// TIA Portal V19 export
VAR_GLOBAL   // PLC tag table "STEP7 classic symbols"
   "hf LyeOnly" AT %I600.1 : Bool;   // info for CIP process (Not used)
   hfOperationsMode AT %IW622 : Int;   // IMA Hassia - operations mode,0=shutdown,1=CIP, 2=SIP,4=Production,8=Adjustments
   prProductAvailableF1 AT %Q608.0 : Bool;   // product for filler 1 is ready
   "A02-ACID CONTAINER EMPTY" AT %M70.1 : Bool;   // ALARM 2
   "A19-TT 01.63 TOO LOW" AT %M72.2 : Bool;   // ALARM 19
   "A36-FB FAULT VALVE 01.15" AT %M74.3 : Bool;   // ALARM 36
   "A55-CIP UNIT OCCUIPED" AT %M76.6 : Bool;   // ALARM 55
   "AutoTT0172/IP0157" AT %M91.0 : Bool;   // REGULATOR TT01.72/IP01.57 IN AUTO MODE
   CIP_Hamba_bit_06 AT %M150.6 : Bool;
   CT_ACID_OK AT %M32.4 : Bool;   // ACID CONCENTRATION WITHIN LIMITS
   "DUMMY TEST AIR" AT %M98.5 : Bool;   // DUMMY TEST AIR SUPPLY
   HSL0165_Proxy AT %M50.1 : Bool;
   P_IP0157 AT %QW274 : Word;   // Steam regulating valve
   "Last Scan Time" AT %MW40 : Int;   // Previous Scan Time
   "M21.1" AT %M21.1 : Bool;
   MY0108 AT %M247.3 : Bool;   // Q 9.3; Output modul 1 Channel 11
   MY0147 AT %M248.7 : Bool;   // Q 20.7; Output modul 2 Channel 7
   MY0911 AT %M253.2 : Bool;
   M_LP_Steam_ON AT %M254.6 : Bool;
   One_shut_on AT %M152.3 : Bool;
   P_PT0167 AT %IW266 : Word;   // Filling pressure
   Product_Route AT %Q41.6 : Bool;   // Hamba
   "R.NOT USED 9" AT %M245.0 : Bool;   // RECIEVE FROM UHT MPI NET, NOT USED
   "S.T.02.TANK PRESELE." AT %M243.5 : Bool;   // TANK 2 PRESELECTED SEND TO UHT FROM TANK 02.00 MPI NET
   "S1 STOP PRODUCTION TANK" AT %M113.1 : Bool;   // STEP 1 STOP PRODUCTION TANK
   "S17 FILLER" AT %M126.1 : Bool;   // STEP 17 FILLER
   "S23 FILLER" AT %M126.7 : Bool;   // STEP 23 FILLER
   "S34 FILLER" AT %M128.2 : Bool;   // STEP 34 FILLER
   "S46 FILLER" AT %M129.6 : Bool;   // STEP 46 FILLER
   "S9 CIP TANK" AT %M119.1 : Bool;   // STEP 9 CIP
   SIP_Hamba_bit_05 AT %M151.5 : Bool;
   ST_CIP_M0139 AT %M138.0 : Bool;   // START CIP PUMP
   Sterilisation_Steam AT %Q41.3 : Bool;   // Hamba
   "T 37 DELAY TT 01.78" AT %T37 : Timer;   // DELAY ALARM TT 01.78 AS BARRIER
   "T53 DETERGENT CONC OK" AT %T53 : Timer;   // DETERGENT CONCENTRATION OK IN X SECONDS
   "TEST BARRIERS" AT %M94.3 : Bool;   // TEST TEMPERATURES AS BARRIERES
   TIM20 AT %M61.2 : Bool;   // START TIMER 20
   TIM37 AT %M63.3 : Bool;   // START TIMER 37
   TIM54 AT %M65.4 : Bool;   // START TIMER 54
   "UHT_STERILE?" AT %I25.5 : Bool;   // UHT STERILE
   Y0104S AT %I12.2 : Bool;   // FEEDBACK SET VALVE 01.04
   Y0114R AT %I16.7 : Bool;   // FEEDBACK RESET VALVE 01.14
   Y0137 AT %Q20.4 : Bool;   // WATER TO CONDENSATER VALVE
   Y0905R AT %I45.1 : Bool;   // On off valve
   Y0910 AT %Q40.6 : Bool;   // Routing valve
   "0.5Hz" AT %M10.7 : Bool;   // CYCLIC CLOCK
   "A04-TANK NOT CLEAN" AT %M70.3 : Bool;   // ALARM 4
   "A21-TT 01.76 LOW" AT %M72.4 : Bool;   // ALARM 21
   "A38-FB FAULT MOTOR 01.30" AT %M74.5 : Bool;   // ALARM 38
   ACID_READY AT %Q29.0 : Bool;   // ACID READY
   ATI AT %M11.2 : Bool;   // Always true input
   "B01.41" AT %I17.4 : Bool;   // HIGH LEVEL ELECTRODE CIP TANK
   CAUSTIC_REQ AT %I33.2 : Bool;   // CAUSTIC REQUIRED
   "CIP_OCCUIPED?" AT %I25.7 : Bool;   // CIP OCCUPIED
   "DUMMY TEST STEAM" AT %M98.4 : Bool;   // DUMMY TEST STEAM SUPPLY
   "I33.7SPARE" AT %I33.7 : Bool;   // SPARE
   M0139 AT %Q9.1 : Bool;   // CIP PUMP
   "M21.3" AT %M21.3 : Bool;   // fp bit for depressurise pg line if not sterile
   MY0111 AT %M246.4 : Bool;   // Q 8.4; Output modul 1 Channel 4
   MY0158 AT %M249.1 : Bool;   // Q 21.1; Output modul 2 Channel 9
   "M_251.3SpareOutput" AT %M251.3 : Bool;   // Q 29.3; Output modul 3 Channel 11
   M_PACK2 AT %M249.4 : Bool;   // Q 21.4; Output modul 2 Channel 12
   Min_F2 AT %IW618 : Word;
   "PULSE 01.13 CIP" AT %M94.6 : Bool;   // PULSE VALVE 01.13 IN CIP
   Prod_Hamba_bit_00 AT %M153.0 : Bool;
   "Q537.0" AT %Q537.0 : Bool;   // Polygon Filler 2 EOL in Use Becon
   "R.UHT STERIL/PRESTE" AT %M244.0 : Bool;   // UHT STERIL/PRESTERIL. RECIEVE FROM UHT MPI NET
   RTE_404_TestBit AT %M19.0 : Bool;   // for testing RTE 404
   "S0 CHAIN WASH" AT %M137.0 : Bool;   // STEP 0 CHAIN WASH
   "S10 CIP TANK" AT %M119.2 : Bool;   // STEP 10 CIP
   "S18 FILLER" AT %M126.2 : Bool;   // STEP 18 FILLER
   "S25 FILLER" AT %M127.1 : Bool;   // STEP 25 FILLER
   "S36 FILLER" AT %M128.4 : Bool;   // STEP 36 FILLER
   "S48 FILLER" AT %M130.0 : Bool;   // STEP 48 FILLER
   SCADA_WD AT %MW200 : Int;   // SCADA Watch Dog
   SIP_Hamba_bit_07 AT %M151.7 : Bool;
   "T 14 STERILE TIME" AT %T14 : Timer;   // STERILIZING TIME ASEPTIC TANK
   "T 39 RUN 01.30" AT %T39 : Timer;   // RUN TIME AGITATOR 01.30
   "T55 ACID DOSING TOO LONG" AT %T55 : Timer;   // ACID DOSING TIME TOO LONG, SEARCH FOR FAILURE
   "TEST FILLING PRESSURE" AT %M94.4 : Bool;   // TEST FILLING PRESSURE
   TIM22 AT %M61.4 : Bool;   // START TIMER 22
   TIM39 AT %M63.5 : Bool;   // START TIMER 39
   TIM56 AT %M65.6 : Bool;   // START TIMER 56
   "UPD.TIMER 14" AT %M84.0 : Bool;   // UPDATE STERILE TIMER
   "V0945-SV2 DelayOff" AT %T77 : Timer;   // V0945-SV2 DelayOff (Production Only)
   WATER_SUPPLY_PUMP AT %Q29.2 : Bool;   // WATER PUMP
   Y0108R AT %I17.3 : Bool;   // FEEDBACK RESET VALVEL 01.08
   Y0115 AT %Q9.0 : Bool;   // WATER TO BALANCE TANK VALVE
   Y0144 AT %Q20.6 : Bool;   // DRAIN VALVE CIP 01.01
   Y0906 AT %Q40.2 : Bool;   // Routing valve
   Y0910S AT %I44.6 : Bool;   // Routing valve
   "hf PreRinse1" AT %I601.0 : Bool;   // prerinse 1
   mw212_DW AT %MW212 : Word;   // Dummy word for fc3
   "hf HoperLevelF1" AT %IW610 : Int;   // Hassia Filler 1 Hopper Level (1000 x 0.1 = 100.0%)
   "hf SIPrequest" AT %I604.0 : Bool;   // request sterilization
   prF2_AhvLevel AT %QW610 : Int;   // Supplying AHV Level for IMA Hassia- Filler2
   "2Hz" AT %M10.3 : Bool;   // CYCLIC CLOCK
   "A14-WAITING FOR CIPUNIT" AT %M71.5 : Bool;   // ALARM 14
   "A31-FB FAULT VALVE 01.09" AT %M73.6 : Bool;   // ALARM 31
   "A48-FB FAULT VALVE 01.19" AT %M75.7 : Bool;   // ALARM 48
   AHV_SHUT_DOWN AT %Q28.3 : Bool;   // AHV SHUT DOWN
   CIP_Hamba_bit_01 AT %M150.1 : Bool;
   "DUMMY 2 FILLING" AT %M100.1 : Bool;   // DUMMY USED IN FILLING
   DisableMonitoringTT0951 AT %M152.2 : Bool;
   "FILLING PIPE DRAINED" AT %M95.2 : Bool;   // FILLING PIPE DRAINED INITIAL START
   GS22_62 AT %I46.1 : Bool;
   "I      47.3" AT %I47.3 : Bool;
   "M20.2" AT %M20.2 : Bool;   // acDataPointer_FIFO #busy in/out
   MW_202 AT %MW202 : Word;
   MY0135 AT %M248.2 : Bool;   // Q 20.2; Output modul 2 Channel 2
   "MY0906 Cycle On" AT %M253.6 : Bool;
   M_Barrier_Sterlising AT %M254.5 : Bool;
   M_WATER_SUPPLY_PUMP AT %M251.2 : Bool;   // Q 29.2; Output modul 3 Channel 10
   PROG_2_SELECTED AT %I32.7 : Bool;   // PROGRAM 2 SELECTED
   Prod_Hamba_bit_10 AT %M154.2 : Bool;
   "R.NOT USED 15" AT %M245.6 : Bool;   // RECIEVE FROM UHT MPI NET, NOT USED
   RINSE_REQ AT %I33.1 : Bool;   // RINSE REQUIRED
   "S.T.02.NOT USED 7" AT %M243.6 : Bool;   // SEND TO UHT FROM TANK 02.00 MPI NET, NOT USED
   "S1 CIP TANK" AT %M118.1 : Bool;   // STEP 1 CIP
   "S15 CIP TANK" AT %M119.7 : Bool;   // STEP 15 CIP
   "S2 TOTAL STOP TANK" AT %M114.2 : Bool;   // STEP 2 TOTAL STOP TANK
   "S3 STOP PRESTE. TANK" AT %M109.3 : Bool;   // STEP 3 STOP PRESTERILIZING TANK
   "S41 FILLER" AT %M129.1 : Bool;   // STEP 41 FILLER
   "S7 CIP TANK" AT %M118.7 : Bool;   // STEP 7 CIP
   SIP_Hamba_bit_00 AT %M151.0 : Bool;
   "Spare m254.7" AT %M254.7 : Bool;
   "T 32 ACID CIRCULATION" AT %T32 : Timer;   // CIRCULATING ACID ASEPTIC TANK
   "T 49 OPEN 01.08 CIP" AT %T49 : Timer;   // OPEN VALVE 01.08 CIP
   "TANK STERILE" AT %M90.2 : Bool;   // TANK IS STERILE
   TIM15 AT %M60.5 : Bool;   // START TIMER 15
   TIM32 AT %M62.6 : Bool;   // START TIMER 32
   TIM49 AT %M64.7 : Bool;   // START TIMER 49
   P_TT0178 AT %IW258 : Word;   // Steam barrier filling valve
   "Trigger bit 4" AT %M14.3 : Bool;   // Trigger bit for calls in item control
   "UPD.TIMER 33" AT %M85.2 : Bool;   // UPDATE WATER 3 TIMER
   ValveHandling3 AT %M3.7 : Bool;   // VALVE HANDLING
   Y0103 AT %Q8.1 : Bool;   // CIP / STEAM INLET VALVE
   Y0112S AT %I12.5 : Bool;   // FEEDBACK SET VALVE 01.12
   Y0119 AT %Q20.0 : Bool;   // FLUSH CHAIN WASH
   Y0904 AT %Q40.0 : Bool;   // On off valve
   "A12-DRAIN TANK NOT ALLOW" AT %M71.3 : Bool;   // ALARM 12
   "A29-FB FAULT VALVE 01.03" AT %M73.4 : Bool;   // ALARM 29
   "A46-FB FAULT VALVE 01.17" AT %M75.5 : Bool;   // ALARM 46
   Barrier_Sterile AT %Q41.5 : Bool;   // Hamba
   DUMMY_ALARM AT %M11.4 : Bool;   // Dummy USED FOR ALARMS ETC
   FILLER_ON_PROD AT %I32.4 : Bool;   // FILLER ON PRODUCT
   "I      47.1" AT %I47.1 : Bool;
   MY0119 AT %M248.0 : Bool;   // Q 20.0; Output modul 2 Channel 0
   MY0905 AT %M252.4 : Bool;
   M_AHV_STERILE AT %M250.4 : Bool;   // Q 28.4; Output modul 3 Channel 4
   M_TANK_READY AT %M251.6 : Bool;   // Q 29.6; Output modul 3 Channel 14
   PROD_AVAILABLE AT %Q28.5 : Bool;   // PRODUCT AVAILABLE
   Prod_Hamba_bit_08 AT %M154.0 : Bool;
   "R.NOT USED 13" AT %M245.4 : Bool;   // RECIEVE FROM UHT MPI NET, NOT USED
   "Request CIP Pump ON" AT %I33.6 : Bool;   // SPARE
   "S.T.01.TANK READY" AT %M242.4 : Bool;   // TANK 1 READY SEND TO UHT FROM TANK 01.00 MPI NET
   "S0 TOTAL STOP TANK" AT %M114.0 : Bool;   // MAIN FLAG TOTAL STOP TANK
   "S14 CIP TANK" AT %M119.6 : Bool;   // STEP 14 CIP
   "S2 STOP PRESTE. TANK" AT %M109.2 : Bool;   // STEP 2 STOP PRESTERILIZING TANK
   "S3 PRESTERILIZING" AT %M110.3 : Bool;   // STEP 3 PRESTERILIZING TANK
   "S4 STOP CIP TANK" AT %M122.4 : Bool;   // STEP 4 STOP CIP
   "S6 FILLER" AT %M124.6 : Bool;   // STEP 06 FILLER
   SIP_Hamba_High_SteamPres AT %M152.0 : Bool;
   "T 30 WATER 2" AT %T30 : Timer;   // INTERMEDIATE RINSE ASEPTIC TANK
   "T 47 OPEN 01.13 PRES" AT %T47 : Timer;   // OPEN TIME VALVE 01.13 IN PRESTERILIZING
   "TANK CLEAN" AT %M0.1 : Bool;   // TANK IS CLEAN
   TIM13 AT %M60.3 : Bool;   // START TIMER 13
   TIM30 AT %M62.4 : Bool;   // START TIMER 30
   TIM47 AT %M64.5 : Bool;   // START TIMER 47
   TIM64 AT %M66.6 : Bool;   // START TIMER 64
   P_TT0172 AT %IW262 : Word;   // CIP temperature
   "Trigger bit 2" AT %M14.1 : Bool;   // Trigger bit for calls in item control
   "UPD.TIMER 31" AT %M85.0 : Bool;   // UPDATE DOSING ACID TIMER
   ValveHandling1 AT %M2.4 : Bool;   // VALVE HANDLING
   Y0101R AT %I16.0 : Bool;   // FEEDBACK RESET VALVE 01.01
   Y0112 AT %Q8.5 : Bool;   // FILLING LINE STOP VALVE
   Y0117S AT %I24.1 : Bool;   // FEEDBACK SET VALVE 01.17
   Y0902 AT %Q29.4 : Bool;   // Low steam pressure
   Y0907S AT %I44.3 : Bool;   // On off valve
   "hf HoperLevelF2" AT %IW612 : Int;   // Hassia Filler 2 Hopper Level (1000 x 0.1 = 100.0%)
   "hf SIPrunning" AT %I604.1 : Bool;   // sterilization is running
   "prLife bit" AT %Q600.0 : Bool;   // check communication (clocked signal 0,5 Hz)
   prEnableCIPValveFlipsF1 AT %Q601.1 : Bool;
   "1HZ_ONESHOT" AT %M11.0 : Bool;
   "A10-TANK IS BEEING FILL." AT %M71.1 : Bool;   // ALARM 10
   "A27-SIEMENS BATTERY LOW" AT %M73.2 : Bool;   // ALARM 27
   "A44-FB FAULT VALVE 02.38" AT %M75.3 : Bool;   // ALARM 44
   AHV_CLOSED AT %Q28.0 : Bool;   // AHV BARRIER CLOSED
   CIP_Running AT %I24.6 : Bool;   // Hamba
   "DUMMY1 DRAIN" AT %M98.7 : Bool;   // DUMMY DRAIN FILLING PIPE
   FILLER_2_OK AT %I32.5 : Bool;   // FILLER 2 BARRIER TEMP. OK
   ForceValves AT %M12.0 : Bool;   // FORCE VALVES TO AUTO
   "I      46.7" AT %I46.7 : Bool;
   MANUAL AT %M3.3 : Bool;   // VALVE HANDLING
   MY0117 AT %M247.4 : Bool;   // Q 9.4; Output modul 1 Channel 12
   MY0903 AT %M252.2 : Bool;
   M_AHV_READY AT %M250.2 : Bool;   // Q 28.2; Output modul 3 Channel 2
   M_Sip_Steam AT %M254.1 : Bool;
   PACK2 AT %Q21.4 : Bool;   // RELAY SIGNAL TO PACKING PRODUCT AVAILA.
   Prod_Hamba_bit_06 AT %M153.6 : Bool;
   "R.NOT USED 11" AT %M245.2 : Bool;   // RECIEVE FROM UHT MPI NET, NOT USED
   "S.T.01.TANK OPEN" AT %M242.3 : Bool;   // TANK 1 OPEN SEND TO UHT FROM TANK 01.00 MPI NET
   "S0 STOP PRESTE. TANK" AT %M109.0 : Bool;   // MAIN FLAG STOP PRESTERILIZING TANK
   "S13 CIP TANK" AT %M119.5 : Bool;   // STEP 13 CIP
   "S2 PRESTERILIZING" AT %M110.2 : Bool;   // STEP 2 PRESTERILIZING TANK
   "S3 CIP TANK" AT %M118.3 : Bool;   // STEP 3 CIP
   "S4 FILLER" AT %M124.4 : Bool;   // STEP 04 FILLER
   "S6 CHAIN WASH" AT %M137.6 : Bool;   // STEP 6 CHAIN WASH
   "T 28 DOSING LYE" AT %T28 : Timer;   // DOSING LYE ASEPTIC TANK
   "T 45 PURGE" AT %T45 : Timer;   // PURGING FILLING PIPE
   T83 AT %T83 : Timer;   // delay close V0945 after flips
   TIM11 AT %M60.1 : Bool;   // START TIMER 11
   TIM28 AT %M62.2 : Bool;   // START TIMER 28
   TIM45 AT %M64.3 : Bool;   // START TIMER 45
   TIM62 AT %M66.4 : Bool;   // START TIMER 62
   TRIGGERBYTE AT %MB14 : Byte;   // USED FOR OUTPUT HANDLER
   "UPD.TIMER 29" AT %M84.6 : Bool;   // UPDATE LYE CIRCULATION TIMER
   X0913 AT %Q41.7 : Bool;   // Cip lamp
   Y0111R AT %I16.4 : Bool;   // FEEDBACK RESET VALVE 01.11
   Y0117 AT %Q9.4 : Bool;   // CIP
   Y0545 AT %Q21.2 : Bool;   // STEAM BY-PASS VALVE REDUCED
   Y0907 AT %Q40.3 : Bool;   // On off valve
   Y0912S AT %I25.3 : Bool;   // SPARE
   "hf DrainMachine" AT %I601.1 : Bool;   // drain machine
   Y0910R AT %I45.6 : Bool;   // Routing valve
   "hf NoTimeStop" AT %I600.4 : Bool;   // no fault and no stop during CIP at Hassia Machine
   mw210_DW AT %MW210 : Word;   // Dummy word for fc3
   prSIPRunningF2 AT %Q604.2 : Bool;   // information product line filler 2 SIP is running
   "A06-NO STEAM" AT %M70.5 : Bool;   // ALARM 6
   "A23-NO WATER" AT %M72.6 : Bool;   // ALARM 23
   "A40-LYE DOSING TOO LONG" AT %M74.7 : Bool;   // ALARM 40
   ACTIVATE AT %M3.4 : Bool;   // VALVE HANDLING
   "B01.65" AT %I17.6 : Bool;   // HIGH LEVEL ELECTRODE STERILE TANK
   CHANGING AT %M2.3 : Bool;   // VALVE HANDLING
   CIP_PROG_2 AT %M135.2 : Bool;   // PROGRAM SELECT 2 CIP FILLER
   "DUMMY TEST TT 01.78" AT %M98.3 : Bool;   // DUMMY TEST TT 01.78 AS BARRIER
   "M21.5" AT %M21.5 : Bool;   // PG line Sterile memory
   MY0113 AT %M246.6 : Bool;   // Q 8.6; Output modul 1 Channel 6
   MY0238 AT %M247.7 : Bool;   // Q 9.7; Output modul 1 Channel 15
   "M_251.5SpareOutput" AT %M251.5 : Bool;   // Q 29.5; Output modul 3 Channel 13
   M_ProdLineBeingCleaned AT %M249.5 : Bool;   // Q 21.5; Output modul 2 Channel 13 was M_PACK3
   Prod_Hamba_bit_02 AT %M153.2 : Bool;
   "R.Acid Level Ok" AT %M244.7 : Bool;   // RECIEVE FROM UHT MPI NET, NOT USED
   RTE_405_TestBit AT %M19.1 : Bool;
   "S.T.01.NOT USED 7" AT %M242.6 : Bool;   // SEND TO UHT FROM TANK 01.00 MPI NET, NOT USED
   "S0 FILLER" AT %M124.0 : Bool;   // STEP 00 MAIN FILLER
   "S11 CIP TANK" AT %M119.3 : Bool;   // STEP 11 CIP
   "S19 FILLER" AT %M126.3 : Bool;   // STEP 19 FILLER
   "S27 FILLER" AT %M127.3 : Bool;   // STEP 27 FILLER
   "S38 FILLER" AT %M128.6 : Bool;   // STEP 38 FILLER
   "S5 CHAIN WASH" AT %M137.5 : Bool;   // STEP 5 CHAIN WASH
   "SPIN 01.30 CIP" AT %M94.5 : Bool;   // SPIN AGITATOR IN CIP
   "T 16 BLOW OUT COND" AT %T16 : Timer;   // BLOW OUT CONDENSATE
   "T 41 DELAY STEAM" AT %T41 : Timer;   // DELAY ALARM STEAM
   "T61 CLOSE Y0101" AT %T61 : Timer;   // DELAY BETWEEN Y0101 AND Y0124 (CLOSE)
   TIM24 AT %M61.6 : Bool;   // START TIMER 24
   TIM41 AT %M63.7 : Bool;   // START TIMER 41
   TIM58 AT %M66.0 : Bool;   // START TIMER 58
   "UPD.TIMER 16" AT %M84.2 : Bool;   // UPDATE BLOW OUT CONDENSATE TIMER
   Y0109 AT %Q8.3 : Bool;   // COOLING WATER TO JACKET VALVE
   Y0115S AT %I13.0 : Bool;   // FEEDBACK SET VALVE 01.15
   Y0148 AT %Q21.0 : Bool;   // STEAM VALVE TO STERILZING
   "hf MachineSterile" AT %I604.2 : Bool;   // machine sterile
   "m20.0" AT %M20.0 : Bool;   // FP
   prSIPRunningF1 AT %Q604.1 : Bool;   // information product line filler 1 SIP is running
   "0.625Hz" AT %M10.6 : Bool;   // CYCLIC CLOCK
   "A05-NO INSTRUMENT AIR" AT %M70.4 : Bool;   // ALARM 5
   "A22-TT 01-78 LOW" AT %M72.5 : Bool;   // ALARM 22
   "A39-TANK READY FOR PROD" AT %M74.6 : Bool;   // ALARM 39
   ACID_REQ AT %I33.3 : Bool;   // ACID REQUIRED
   AcidCipPressure AT %M96.3 : Bool;
   "B01.42" AT %I17.5 : Bool;   // LOW LEVEL ELECTRODE CIP TANK
   CHAIN_WASH AT %I33.4 : Bool;   // CHAIN WASH
   CIP_PROG_1 AT %M135.1 : Bool;   // PROGRAM SELECT 1 CIP FILLER
   "DUMMY TEST TT 01.76" AT %M98.2 : Bool;   // DUMMY TEST TT 01.76 AS BARRIER
   "Hamba FP1 Route OK" AT %M104.1 : Bool;
   "I553.0" AT %I533.0 : Bool;   // M0941 - Running (M0940 Cooling Fan)
   Init_Scan AT %M0.0 : Bool;   // First Scan
   M0139S AT %I13.1 : Bool;   // FEEDBACK MOTOR 01.39 RUNNING
   "M21.4" AT %M21.4 : Bool;   // depressurise pg line if clean not sterile
   MY0112 AT %M246.5 : Bool;   // Q 8.5; Output modul 1 Channel 5
   MY0237 AT %M247.6 : Bool;   // Q 9.6; Output modul 1 Channel 14
   "M_251.4SpareOutput" AT %M251.4 : Bool;   // Q 29.4; Output modul 3 Channel 12
   M_PROD_AVAILABLE AT %M250.5 : Bool;   // Q 28.5; Output modul 3 Channel 5
   "PULSE 01.18 PRESTERILI" AT %M94.0 : Bool;   // PULSING VALVE 01.13 IN PRESTERILIZING
   Prod_Hamba_bit_01 AT %M153.1 : Bool;
   "Q537.1" AT %Q537.1 : Bool;   // Polygon F2 Product at Filler
   "S.T.01.ALARM PULS" AT %M242.2 : Bool;   // ALARM PULS SEND TO UHT FROM TANK 01.00 MPI NET
   "S0 CIP TANK" AT %M118.0 : Bool;   // MAIN FLAG CIP
   "S10 FILLER" AT %M125.2 : Bool;   // STEP 10 FILLER
   "S19 CIP TANK" AT %M120.3 : Bool;   // STEP 19 CIP
   "S26 FILLER" AT %M127.2 : Bool;   // STEP 26 FILLER
   "S37 FILLER" AT %M128.5 : Bool;   // STEP 37 FILLER
   "S49 FILLER" AT %M130.1 : Bool;   // STEP 49 FILLER
   "SOFTKEY 5 DRAIN TANK" AT %M99.6 : Bool;   // SOFTKEY START DRAIN TANK
   "T 15 COOLING TIME" AT %T15 : Timer;   // COOLING TIME ASEPTIC TANK
   "T 40 RESET STOP LIGHT" AT %T40 : Timer;   // DELAY RESET STOP LIGHT AFTER 3 SEC
   "T60 OPEN Y0101" AT %T60 : Timer;   // DELAY BETWEEN Y0124 AND Y0101 (OPEN)
   TIM23 AT %M61.5 : Bool;   // START TIMER 23
   TIM40 AT %M63.6 : Bool;   // START TIMER 40
   TIM57 AT %M65.7 : Bool;   // START TIMER 57
   "UPD.TIMER 15" AT %M84.1 : Bool;   // UPDATE COOLING TIMER
   Y0108S AT %I13.3 : Bool;   // FEEDBACK SET VALVEL 01.18
   Y0115R AT %I17.0 : Bool;   // FEEDBACK RESET VALVE 01.15
   Y0147 AT %Q20.7 : Bool;   // STEAM VALVE TO 01.13
   "Y0906 Cycle Off" AT %M253.7 : Bool;
   Y0911 AT %Q40.7 : Bool;   // On off valve
   "A01-LYE CONTAINER EMPTY" AT %M70.0 : Bool;   // ALARM 1
   "A18-TT 01.60 TOO LOW" AT %M72.1 : Bool;   // ALARM 18
   "A35-FB FAULT VALVE 01.14" AT %M74.2 : Bool;   // ALARM 35
   "A54-NO CIP PROG SEL" AT %M76.5 : Bool;   // ALARM 54
   "AutoPT0167/IP0149" AT %M91.2 : Bool;   // REGULATOR PT01.67/IP01.49 IN AUTO MODE
   CIP_Hamba_bit_05 AT %M150.5 : Bool;
   P_CT0182 AT %IW270 : Word;   // CIP Contration return
   "DUMMY START AGITATOR" AT %M99.3 : Bool;   // DUMMY START AGITATOR
   "FS01.81" AT %I13.2 : Bool;   // FLOW SWITCH CIP RETURN
   "I      47.7" AT %I47.7 : Bool;
   P_IP014950 AT %QW272 : Word;   // Sterile air control valves
   "M21.0" AT %M21.0 : Bool;
   MY0104 AT %M246.2 : Bool;   // Q 8.2; Output modul 1 Channel 2
   MY0144 AT %M248.6 : Bool;   // Q 20.6; Output modul 2 Channel 6
   MY0910 AT %M253.1 : Bool;
   M_Cip_Route AT %M254.0 : Bool;
   Max_F2 AT %IW620 : Word;
   One_shut_off AT %M152.4 : Bool;
   Product_Request AT %I24.5 : Bool;   // Hamba
   "R.NOT USED 6" AT %M244.5 : Bool;   // RECIEVE FROM UHT MPI NET, NOT USED
   RTE_404_Cip_Route_Open AT %M255.0 : Bool;   // Allow Gemini Route 411 and Tankroom Route 404_405 to Run
   "S.T.02.TANK OPEN" AT %M243.3 : Bool;   // TANK 2 OPEN SEND TO UHT FROM TANK 02.00 MPI NET
   "S1 STOP PRESTE. TANK" AT %M109.1 : Bool;   // STEP 1 STOP PRESTERILIZING TANK
   "S17 CIP TANK" AT %M120.1 : Bool;   // STEP 17 CIP
   "S22 FILLER" AT %M126.6 : Bool;   // STEP 22 FILLER
   "S33 FILLER" AT %M128.1 : Bool;   // STEP 33 FILLER
   "S45 FILLER" AT %M129.5 : Bool;   // STEP 45 FILLER
   "S8 FILLER" AT %M125.0 : Bool;   // STEP 08 FILLER
   SIP_Hamba_bit_04 AT %M151.4 : Bool;
   StepOldStatus AT %MW208 : Word;   // Dummy word for fc3
   "T 36 DELAY TT 01.76" AT %T36 : Timer;   // DELAY ALARM TT 01.76 AS BARRIER
   T20_Trigger_bit AT %T20 : Timer;
   "TBM DUMMY MOTOR 01.39" AT %M79.0 : Bool;   // DUMMY FEED-BACK FOR RESET
   TIM19 AT %M61.1 : Bool;   // START TIMER 19
   TIM36 AT %M63.2 : Bool;   // START TIMER 36
   TIM53 AT %M65.3 : Bool;   // START TIMER 53
   "Trigger bit 8" AT %M14.7 : Bool;   // Trigger bit for calls in item control
   UnforceValves AT %M12.1 : Bool;   // UNFORCE VALVES FROM AUTO
   Y0104R AT %I16.2 : Bool;   // FEEDBACK RESET VALVE 01.04
   Y0114 AT %Q8.7 : Bool;   // CIP RETURN / DRAIN VALVE
   Y0136 AT %Q20.3 : Bool;   // STEAM TO CONDENSTATE VALVE
   Y0905 AT %Q40.1 : Bool;   // On off valve
   Y0909S AT %I44.5 : Bool;   // On off valve
   "hf MachineIsClean" AT %I601.7 : Bool;   // machine is clean
   "m19.3" AT %M19.3 : Bool;   // Tank Sterile for testing
   prReadyForCIP AT %Q600.1 : Bool;
   "Y0906 Cycle Off Timer" AT %T66 : Timer;
   Y0911R AT %I45.7 : Bool;   // On off valve
   "hf AcidCirculation" AT %I601.5 : Bool;   // cycle acid
   "hf ProductPumpRequestF1" AT %I608.1 : Bool;   // start product pump filler 1
   prEnableCIPReturnPump AT %Q600.3 : Bool;
   "1HZ" AT %M10.5 : Bool;   // CYCLIC CLOCK
   "A09-ALREADY IN STOP" AT %M71.0 : Bool;   // ALARM 9
   "A26-TANK FULL" AT %M73.1 : Bool;   // ALARM 26
   "A43-FB FAULT VALVE 02.37" AT %M75.2 : Bool;   // ALARM 43
   "AGITATOR MANUEL" AT %M95.1 : Bool;   // AGITATOR IN MANUEL MODE
   Alarm_battery_low_dummy AT %M7.0 : Bool;
   "B02.77" AT %I17.2 : Bool;   // ACID LEVEL IN ACID CONTAINER
   CIP_Route_Request AT %I24.3 : Bool;   // Hamba
   "DUMMY UPD.DRAIN TANK" AT %M99.7 : Bool;   // UPDATING DRAIN TANK ACTIVATED
   Flow_Pulse_Mem AT %M2.0 : Bool;
   "I      46.6" AT %I46.6 : Bool;
   "M22.0" AT %M22.0 : Bool;   // M0940 Pump Casing < 70°C
   MY0116 AT %M247.2 : Bool;   // Q 9.2; Output modul 1 Channel 10
   MY0902 AT %M252.1 : Bool;
   M_AHV_HIGH_LEVEL AT %M250.1 : Bool;   // Q 28.1; Output modul 3 Channel 1
   M_RINSE_READY AT %M250.6 : Bool;   // Q 28.6; Output modul 3 Channel 6
   PACK1 AT %Q21.3 : Bool;   // RELAY SIGNAL TO PACKING PRODUCT AVAILA.
   Prod_Hamba_bit_05 AT %M153.5 : Bool;
   "R.NOT USED 10" AT %M245.1 : Bool;   // RECIEVE FROM UHT MPI NET, NOT USED
   "S.T.01.REQUEST LYE" AT %M242.0 : Bool;   // REQUEST LYE SEND TO UHT FROM TANK 01.00 MPI NET
   "S0 STOP CIP TANK" AT %M122.0 : Bool;   // MAIN FLAG STOP CIP
   "S12 FILLER" AT %M125.4 : Bool;   // STEP 12 FILLER
   "S2 FILLER" AT %M124.2 : Bool;   // STEP 02 FILLER
   "S3 CHAIN WASH" AT %M137.3 : Bool;   // STEP 3 CHAIN WASH
   "S4 CIP TANK" AT %M118.4 : Bool;   // STEP 4 CIP
   "S5 PRESTERILIZING" AT %M110.5 : Bool;   // STEP 5 PRESTERILIZING TANK
   Set_alarm_lamp_process AT %M6.2 : Bool;
   "T 27 WATER 1" AT %T27 : Timer;   // PRERINSE ASEPTIC TANK
   "T 44 FILLING DRAIN" AT %T44 : Timer;   // DELAY BEFORE PURGING
   T75 AT %T75 : Timer;   // M0940 - Wait to cool
   TIM10 AT %M60.0 : Bool;   // START TIMER 10
   TIM27 AT %M62.1 : Bool;   // START TIMER 27
   TIM44 AT %M64.2 : Bool;   // START TIMER 44
   TIM61 AT %M66.3 : Bool;   // START TIMER 61
   "Time Stop CIP" AT %Q21.6 : Bool;   // Signal to Combi 512
   "UPD.TIMER 28" AT %M84.5 : Bool;   // UPDATE DOSING LYE TIMER
   VLV_ALARM AT %M2.5 : Bool;   // VALVE HANDLING
   WaterPumpS AT %I13.6 : Bool;   // FEEDBACK WATER SUPPLY PUMP
   Y0111 AT %Q8.4 : Bool;   // STERILE AIR INLET VALVE
   Y0116S AT %I24.0 : Bool;   // FEEDBACK SET VALVE 01.16
   Y0238 AT %Q9.7 : Bool;   // RELAY SIGNAL TO UHT REQUEST ACID
   Y0906S AT %I44.2 : Bool;   // Routing valve
   Y0912R AT %I25.4 : Bool;   // SPARE
   "hf CIPrunning" AT %I600.3 : Bool;   // CIP is running at Hassia Machine
   "hf ProductRequestF2" AT %I609.0 : Bool;   // request product filler 2
   prEnableSIP AT %Q604.0 : Bool;
   steam_lp_enabled AT %Q41.1 : Bool;
   delayResetOfObjEn AT %T70 : Timer;   // Delay reset of CC_CL_ObjEn
   "hf PreRinse2" AT %I601.2 : Bool;   // prerinse 2
   prCIPStepEnable AT %Q600.4 : Bool;   // medium OK mean: flow OK, conductivity OK and temperatur OK
   prSterileF2 AT %Q604.4 : Bool;   // product line filler 2 is sterilized (ready for production)
   "10Hz" AT %M10.0 : Bool;   // CYCLIC CLOCK
   "A08-NO PROCESS ACTIVE" AT %M70.7 : Bool;   // ALARM 8
   "A25-TANK EMPTY" AT %M73.0 : Bool;   // ALARM 25
   "A42-DRAIN IS ACTIVE" AT %M75.1 : Bool;   // ALARM 42
   "AGITATOR AUTOMATIC" AT %M95.0 : Bool;   // AGITATOR IN AUTOMATIC MODE
   "B02.76" AT %I17.1 : Bool;   // LYE LEVEL IN LYE CONTAINER
   "CIP Stop Push Button" AT %I24.7 : Bool;   // CIP Stop Request for Hambra
   CIP_Route AT %Q41.2 : Bool;   // Hamba
   "DUMMY TEST WATER" AT %M98.6 : Bool;   // DUMMY TEST WATER SUPPLY
   "I      46.5" AT %I46.5 : Bool;
   "INPUT SET" AT %M2.1 : Bool;
   "M21.7" AT %M21.7 : Bool;   // M0940 Activated Memory
   MY0115 AT %M247.0 : Bool;   // Q 9.0; Output modul 1 Channel 8
   MY0901 AT %M252.0 : Bool;
   M_AHV_CLOSED AT %M250.0 : Bool;   // Q 28.0; Output modul 3 Channel 0
   M_Product_Route AT %M254.4 : Bool;
   PA0572_Air AT %I13.5 : Bool;   // PRESSOSTAT FOR INSTRUMENT AIR NC
   Prod_Hamba_bit_04 AT %M153.4 : Bool;
   "R.Lye Level Ok" AT %M244.6 : Bool;   // RECIEVE FROM UHT MPI NET, NOT USED
   RTE_406_TestBit AT %M19.2 : Bool;
   "S.T.01.REQUEST ACID" AT %M242.1 : Bool;   // REQUEST ACID SEND TO UHT FROM TANK 01.00 MPI NET
   "S0 PRODUCTION TANK" AT %M112.0 : Bool;   // MAIN FLAG PRODUCTION TANK
   "S12 CIP TANK" AT %M119.4 : Bool;   // STEP 12 CIP
   "S2 CIP TANK" AT %M118.2 : Bool;   // STEP 2 CIP
   "S29 FILLER" AT %M127.5 : Bool;   // STEP 29 FILLER
   "S4 CHAIN WASH" AT %M137.4 : Bool;   // STEP 4 CHAIN WASH
   "S5 FILLER" AT %M124.5 : Bool;   // STEP 05 FILLER
   "START FILLING TANK" AT %M112.1 : Bool;
   Set_alarm_lamp_monitor AT %M6.1 : Bool;
   "T 18 DELAY 01.12" AT %T18 : Timer;   // DELAY OPEN 01.12
   "T 43 DELAY WATER" AT %T43 : Timer;   // DELAY ALARM WATER
   T74 AT %T74 : Timer;   // PG F2 Prod At Filler signal delay Off.
   TIM26 AT %M62.0 : Bool;   // START TIMER 26
   TIM43 AT %M64.1 : Bool;   // START TIMER 43
   TIM60 AT %M66.2 : Bool;   // START TIMER 60
   "UPD.TIMER 27" AT %M84.4 : Bool;   // UPDATE WATER 1 TIMER
   P_WT0169_TX AT %QW276 : Word;   // Content aseptic tank (Retransmit to Product Transfer System)
   Y0109S AT %I12.3 : Bool;   // FEEDBACK SET VALVE 01.09
   Y0116R AT %I25.0 : Bool;   // FEEDBACK RESET VALVE 01.16
   Y0237 AT %Q9.6 : Bool;   // RELAY SIGNAL TO UHT REQUEST LYE
   Y0906R AT %I45.2 : Bool;   // Routing valve
   Y0912 AT %Q41.0 : Bool;   // Routing valve
   prSterileF1 AT %Q604.3 : Bool;   // product line filler 1 is sterilized (ready for production)
   "1.25Hz" AT %M10.4 : Bool;   // CYCLIC CLOCK
   "A07-NOT READY FOR CIP" AT %M70.6 : Bool;   // ALARM 7
   "A24-PRODUCT AT FILLING" AT %M72.7 : Bool;   // ALARM 24
   "A41-ACID DOSING TOO LONG" AT %M75.0 : Bool;   // ALARM 41
   AFI AT %M11.3 : Bool;   // Always false input
   "B01.66" AT %I17.7 : Bool;   // LOW LEVEL ELECTRODE STERILE TANK
   "CIP Release" AT %Q21.7 : Bool;   // Signal to Combi 512
   CIP_PROG_3 AT %M135.3 : Bool;   // PROGRAM SELECT 3 CIP FILLER
   "DUMMY TEST TT 09.51" AT %M97.0 : Bool;   // DUMMY TEST TT 09.51 AS BARRIER
   "I      46.4" AT %I46.4 : Bool;
   INIT_1HZ_ONESHOT AT %M11.1 : Bool;
   "M21.6" AT %M21.6 : Bool;   // M0940 Activated Memory FP
   MY0114 AT %M246.7 : Bool;   // Q 8.7; Output modul 1 Channel 7
   MY0545 AT %M249.2 : Bool;   // Q 21.2; Output modul 2 Channel 10
   M_ACID_READY AT %M251.0 : Bool;   // Q 29.0; Output modul 3 Channel 8
   M_Product_Available AT %M254.2 : Bool;
   PA0561_Steam AT %I13.4 : Bool;   // PRESSOSTAT FOR STEAM NO
   Prod_Hamba_bit_03 AT %M153.3 : Bool;
   "R.CIP UNIT OCCUPIED" AT %M244.2 : Bool;   // CIP UNIT OCCUPIED. RECIEVE FROM UHT MPI NET
   "S.T.01.NOT USED 8" AT %M242.7 : Bool;   // SEND TO UHT FROM TANK 01.00 MPI NET, NOT USED
   "S0 PRESTERILIZING" AT %M110.0 : Bool;   // MAIN FLAG PRESTERILIZING TANK
   "S11 FILLER" AT %M125.3 : Bool;   // STEP 11 FILLER
   "S2 CHAIN WASH" AT %M137.2 : Bool;   // STEP 2 CHAIN WASH
   "S28 FILLER" AT %M127.4 : Bool;   // STEP 28FILLER
   "S39 FILLER" AT %M128.7 : Bool;   // STEP 39 FILLER
   "S5 CIP TANK" AT %M118.5 : Bool;   // STEP 5 CIP
   "SPIN 01.30 PRESTERILI" AT %M94.1 : Bool;   // SPIN AGITATOR 01.30 IN PRESTERILIZING
   Set_alarm_lamp_feedback AT %M6.0 : Bool;
   "T 17 BLOW OUT STOP" AT %T17 : Timer;   // BLOW OUT AFTER STOP
   "T 42 DELAY AIR" AT %T42 : Timer;   // DELAY ALARM AIR
   T73 AT %T73 : Timer;   // PG F2 Prod At Filler signal delay On.
   "TEST TEMPS. PRESTERILI" AT %M94.2 : Bool;   // TEST TEMEPERATURES IN PRESTERILIZNG
   TIM25 AT %M61.7 : Bool;   // START TIMER 25
   TIM42 AT %M64.0 : Bool;   // START TIMER 42
   TIM59 AT %M66.1 : Bool;   // START TIMER 59
   "UPD.TIMER 17" AT %M84.3 : Bool;   // UPDATE BLOW OUT STOP TIMER
   P_WT0169 AT %IW268 : Word;   // Content aseptic tank
   Y0109R AT %I16.3 : Bool;   // FEEDBACK RESET VALVE 01.09
   Y0116 AT %Q9.2 : Bool;   // CIP RETURN FROM TANK/FILLING
   Y0158 AT %Q21.1 : Bool;   // STEAM VALVE TO INJECTOR
   "Y0906 Cycle On Timer" AT %T67 : Timer;
   Y0911S AT %I44.7 : Bool;   // On off valve
   "hf AcidRinse" AT %I601.6 : Bool;   // clear rinse after acid
   "hf ProductPumpRequestF2" AT %I609.1 : Bool;   // start product pump filler 2
   Y0908R AT %I45.4 : Bool;   // On off valve
   "hf LyeAcid" AT %I600.2 : Bool;   // info for CIP process (Not used)
   "hf SteamBarrierActiveF2" AT %I605.1 : Bool;   // steam barrier valve cluster filler 2 active
   prProdLineCIPRunningF1 AT %Q601.0 : Bool;
   "5Hz" AT %M10.1 : Bool;   // CYCLIC CLOCK
   "A17-TT 01.76 TOO LOW" AT %M72.0 : Bool;   // ALARM 17
   "A34-FB FAULT VALVE 01.13" AT %M74.1 : Bool;   // ALARM 34
   "A53-CHAIN WASH SELECTED" AT %M76.4 : Bool;   // ALARM 53
   ALR_COUNT AT %M2.6 : Bool;   // VALVE HANDLING
   CIP_Hamba_bit_04 AT %M150.4 : Bool;
   "Continue_in program" AT %M96.1 : Bool;
   "DUMMY RESET TANK" AT %M98.0 : Bool;   // DUMMY RESET ALL TANK
   "FORCE ON" AT %M3.0 : Bool;   // VALVE HANDLING
   "Gasti FP1 Route OK" AT %M104.2 : Bool;
   "I      47.6" AT %I47.6 : Bool;
   "M20.7" AT %M20.7 : Bool;   // Fill to Tank Expired Memory
   MY0103 AT %M246.1 : Bool;   // Q 8.1; Output modul 1 Channel 1
   MY0143 AT %M248.5 : Bool;   // Q 20.5; Output modul 2 Channel 5
   MY0909 AT %M253.0 : Bool;
   M_CIP_FILLER_READY AT %M251.1 : Bool;   // Q 29.1; Output modul 3 Channel 9
   Max_F1 AT %IW616 : Word;
   OUTPUT AT %M2.2 : Bool;
   Product_Available AT %Q41.4 : Bool;   // Hamba
   "R.NOT USED 5" AT %M244.4 : Bool;   // RECIEVE FROM UHT MPI NET, NOT USED
   RTE406_MSG AT %T92 : Timer;   // Route 406 Message Display Timer
   "S.T.02.REQUEST LYE" AT %M243.0 : Bool;   // REQUEST LYE SEND TO UHT FROM TANK 02.00 MPI NET
   "S1 STOP CIP TANK" AT %M122.1 : Bool;   // STEP 1 STOP CIP
   "S16 FILLER" AT %M126.0 : Bool;   // STEP 16 FILLER
   "S21 FILLER" AT %M126.5 : Bool;   // STEP 21 FILLER
   "S32 FILLER" AT %M128.0 : Bool;   // STEP 32 FILLER
   "S44 FILLER" AT %M129.4 : Bool;   // STEP 44FILLER
   "S8 CIP TANK" AT %M119.0 : Bool;   // STEP 8 CIP
   SIP_Hamba_bit_03 AT %M151.3 : Bool;
   Steam_Request AT %I24.4 : Bool;   // Hamba
   "T 35 DELAY PT 01.67" AT %T35 : Timer;   // DELAY ALARM FILLING PRESSURE
   "T 52 FLIP 01.44" AT %T52 : Timer;   // FLIP VALVE 01.44 AT STOP FILLING
   "TBM DUMMY MOTOR 01.30" AT %M79.1 : Bool;   // DUMMY FEED-BACK FOR RESET
   TIM18 AT %M61.0 : Bool;   // START TIMER 18
   TIM35 AT %M63.1 : Bool;   // START TIMER 35
   TIM52 AT %M65.2 : Bool;   // START TIMER 52
   P_TT0951 AT %IW402 : Word;   // Steam barrier temperature
   "Trigger bit 7" AT %M14.6 : Bool;   // Trigger bit for calls in item control
   "UPD.TIMER 39" AT %M85.5 : Bool;   // UPDATE RUN TIMER AGITATOR
   Y0104 AT %Q8.2 : Bool;   // CIP / STEAM INLET VALVE
   Y0113S AT %I12.6 : Bool;   // FEEDBACK SET VALVE 01.13
   Y0135 AT %Q20.2 : Bool;   // CONDENSATE VALVE AGITATOR
   Y0904S AT %I44.0 : Bool;   // On off valve
   "hf LifeBit" AT %I600.0 : Bool;   // Hassia Filler Life Bit to Check Communication ( clocked signal 0.5 Hz)
   "hf SteamBarrierActiveF1" AT %I605.0 : Bool;   // steam barrier valve cluster filler 1 active
   prNoTimeStop AT %Q600.2 : Bool;   // no fault and no stop during CIP at CIP process
   "A16-FILLING PRESSURE LOW" AT %M71.7 : Bool;   // ALARM 16
   "A33-FB FAULT VALVE 01.12" AT %M74.0 : Bool;   // ALARM 33
   "A52-CIP TANK RUNNING" AT %M76.3 : Bool;   // ALARM 52
   CIP_Hamba_bit_03 AT %M150.3 : Bool;
   "DUMMY PRODUCT AT TANK" AT %M99.2 : Bool;   // DUMMY PRODUCT AT TANK
   "FORCE OFF" AT %M3.1 : Bool;   // VALVE HANDLING
   GS22_68 AT %I46.3 : Bool;
   "I      47.5" AT %I47.5 : Bool;
   "M20.4" AT %M20.4 : Bool;   // Wait for Process of all Items in reqArrDB
   MY0101 AT %M246.0 : Bool;   // Q 8.0; Output modul 1 Channel 0
   MY0137 AT %M248.4 : Bool;   // Q 20.4; Output modul 2 Channel 4
   MY0908 AT %M252.7 : Bool;
   "M_CIP Release" AT %M249.7 : Bool;   // Q 21.7; Output modul 2 Channel 15
   "ManTT0172/IP0157" AT %M91.1 : Bool;   // REGULATOR TT01.72/IP01.57 IN MANUEL MODE
   Prod_Hamba_bit_12 AT %M154.4 : Bool;
   "R.NOT USED 4" AT %M244.3 : Bool;   // RECIEVE FROM UHT MPI NET, NOT USED
   RTE405_MSG AT %T91 : Timer;   // Route 405 Message Display Timer
   "S.T.02.REQUEST ACID" AT %M243.1 : Bool;   // REQUEST ACID SEND TO UHT FROM TANK 02.00 MPI NET
   "S1 PRESTERILIZING" AT %M110.1 : Bool;   // STEP 1 PRESTERILIZING TANK
   "S16 CIP TANK" AT %M120.0 : Bool;   // STEP 16 CIP
   "S20 FILLER" AT %M126.4 : Bool;   // STEP 20 FILLER
   "S31 FILLER" AT %M127.7 : Bool;   // STEP 31 FILLER
   "S43 FILLER" AT %M129.3 : Bool;   // STEP 43 FILLER
   "S7 PRESTERILIZING" AT %M110.7 : Bool;   // STEP 7 PRESTERILIZING TANK
   SIP_Hamba_bit_02 AT %M151.2 : Bool;
   "T 34 BLOW OUT CIP" AT %T34 : Timer;   // BLOW OUT AFTER CIP
   "T 51 PAUSE 01.08 CIP" AT %T51 : Timer;   // PAUSE TIME BEFORE 01.80 OPEN
   TANK_READY AT %Q29.6 : Bool;   // SIGNAL TO UHT TANK READY
   TIM17 AT %M60.7 : Bool;   // START TIMER 17
   TIM34 AT %M63.0 : Bool;   // START TIMER 34
   TIM51 AT %M65.1 : Bool;   // START TIMER 51
   P_TT0950 AT %IW400 : Word;   // Steam barrier temperature
   "Trigger bit 6" AT %M14.5 : Bool;   // Trigger bit for calls in item control
   "UPD.TIMER 38" AT %M85.4 : Bool;   // UPDATE PAUSE TIMER AGITATOR
   Y0103S AT %I12.1 : Bool;   // FEEDBACK SET VALVE 01.03
   Y0113R AT %I16.6 : Bool;   // FEEDBACK RESET VALVE 01.13
   Y0124 AT %Q20.1 : Bool;   // BY-PASS VALVE STEAM VALVE 01.01
   Y0904R AT %I45.0 : Bool;   // On off valve
   Y0909 AT %Q40.5 : Bool;   // On off valve
   "A15-FILLING PRESSURE TOO" AT %M71.6 : Bool;   // ALARM 15
   "A32-FB FAULT VALVE 01.11" AT %M73.7 : Bool;   // ALARM 32
   "A51-FILLER NOT READY" AT %M76.2 : Bool;   // ALARM 51
   AHV_STERILE AT %Q28.4 : Bool;   // AHV STERILE
   CIP_Hamba_bit_02 AT %M150.2 : Bool;
   "CONTROL CIP TANK" AT %M94.7 : Bool;   // CONTROL LEVEL IN CIP TANK
   "Combi 512 In USE" AT %I32.1 : Bool;   // OSCILLATING SUPPLY SIGNAL
   "DUMMY PROD. AT FILLING" AT %M99.1 : Bool;   // DUMMY PRODUCT AT FILLING MASHINES
   "Dummy Start CIP timer" AT %M96.2 : Bool;
   "FLIP 01.44" AT %M95.4 : Bool;   // FLIP VALVE 01.44 AT STOP FILLING
   GS22_63 AT %I46.2 : Bool;
   "I      47.4" AT %I47.4 : Bool;
   "M20.3" AT %M20.3 : Bool;   // IO-Link Acyclic FP
   MX0913 AT %M253.4 : Bool;
   MY0136 AT %M248.3 : Bool;   // Q 20.3; Output modul 2 Channel 3
   MY0907 AT %M252.6 : Bool;
   M_CAUSTIC_READY AT %M250.7 : Bool;   // Q 28.7; Output modul 3 Channel 7
   "ManPT0167/IP0149" AT %M91.3 : Bool;   // REGULATOR PT01.67/IP01.49 IN MANUEL MODE
   PROG_3_SELECTED AT %I33.0 : Bool;   // PROGRAM 3 SELECTED
   "Polygon FP1 Route OK" AT %M104.0 : Bool;
   Prod_Hamba_bit_11 AT %M154.3 : Bool;
   "R.NOT USED 16" AT %M245.7 : Bool;   // RECIEVE FROM UHT MPI NET, NOT USED
   RTE404_MSG AT %T90 : Timer;   // Route 404 Message Display Timer
   "S.T.02.NOT USED 8" AT %M243.7 : Bool;   // SEND TO UHT FROM TANK 02.00 MPI NET, NOT USED
   "S1 FILLER" AT %M124.1 : Bool;   // STEP 01 FILLER
   "S15 FILLER" AT %M125.7 : Bool;   // STEP 15 FILLER
   "S20 CIP TANK" AT %M120.4 : Bool;   // STEP 20 CIP
   "S30 FILLER" AT %M127.6 : Bool;   // STEP 30 FILLER
   "S42 FILLER" AT %M129.2 : Bool;   // STEP 42 FILLER
   "S7 FILLER" AT %M124.7 : Bool;   // STEP 07 FILLER
   SIP_Hamba_bit_01 AT %M151.1 : Bool;
   "STOP FILLING TANK" AT %M112.2 : Bool;
   "T 33 WATER 3" AT %T33 : Timer;   // FINAL RINSE ASEPTIC TANK
   "T 50 OPEN 01.24 CIP" AT %T50 : Timer;   // OPEN VALVE 01.24 CIP 1/2 TIME T 49
   TANK_OPEN AT %Q29.7 : Bool;   // SIGNAL TO UHT TANK OPEN
   TIM16 AT %M60.6 : Bool;   // START TIMER 16
   TIM33 AT %M62.7 : Bool;   // START TIMER 33
   TIM50 AT %M65.0 : Bool;   // START TIMER 50
   P_TT0180 AT %IW264 : Word;   // CIP return temperature
   "Trigger bit 5" AT %M14.4 : Bool;   // Trigger bit for calls in item control
   "UPD.TIMER 34" AT %M85.3 : Bool;   // UPDATE BLOW OUT CIP TIMER
   Y0103R AT %I16.1 : Bool;   // FEEDBACK RESET VALVE 01.03
   Y0113 AT %Q8.6 : Bool;   // FILLING LINE STEAM / CIP VALVE
   Y0119S AT %I24.2 : Bool;   // FEEDBACK SET VALVE 01.18
   "Y0904-0906_CIP" AT %M253.5 : Bool;
   Y0908S AT %I44.4 : Bool;   // On off valve
   "hf LyeCirculation" AT %I601.3 : Bool;   // cycle caustic
   hfGoodPotCount AT %ID624 : DInt;   // IMA Hassia - Good Pot Count
   prProdLineCIPRunningF2 AT %Q601.2 : Bool;
   Y0909R AT %I45.5 : Bool;   // On off valve
   "hf LyeRinse" AT %I601.4 : Bool;   // clear rinse after caustic
   prProductAvailableF2 AT %Q609.0 : Bool;   // product for filler 2 is ready
   "A03-TANK IN PROCESS" AT %M70.2 : Bool;   // ALARM 3
   "A20-TT 01.78 TOO LOW" AT %M72.3 : Bool;   // ALARM 20
   "A37-FB FAULT MOTOR 01.39" AT %M74.4 : Bool;   // ALARM 37
   "A56-CIP FILLER STARTED" AT %M76.7 : Bool;   // ALARM 56
   CAUSTIC_READY AT %Q28.7 : Bool;   // CAUSTIC READY
   CIP_Hamba_bit_07 AT %M150.7 : Bool;
   CT_LYE_OK AT %M32.3 : Bool;   // LYE CONCENTRATION REACHED SETPOINT
   "DUMMY TEST PT 01.67" AT %M98.1 : Bool;   // DUMMY TEST FILLING PRESSURE
   LowCIPPressure AT %M96.0 : Bool;
   "M21.2" AT %M21.2 : Bool;   // M0940 Condensate OK
   MY0109 AT %M246.3 : Bool;   // Q 8.3; Output modul 1 Channel 3
   MY0148 AT %M249.0 : Bool;   // Q 21.0; Output modul 2 Channel 8
   MY0912 AT %M253.3 : Bool;
   M_PACK1 AT %M249.3 : Bool;   // Q 21.3; Output modul 2 Channel 11
   Min_F1 AT %IW614 : Word;
   "PULSE 01.08 CIP" AT %M95.3 : Bool;   // PULSE VALVE 01.08/01.24 IN CIP
   ProdLineBeingCleaned AT %Q21.5 : Bool;   // Signal to Combi 512
   "Pulse_ FT01.83" AT %I13.7 : Bool;   // FEEDBACK SET M02.38
   "R.PROD  AT TANK" AT %M244.1 : Bool;   // PRODUCTION AT TANK . RECIEVE FROM UHT MPI NET
   RTE_404_Sip_Steam AT %M255.1 : Bool;   // No Return Flow signal to Tankroom Via Gemini
   "S.T.02.TANK READY" AT %M243.4 : Bool;   // TANK 2 READY SEND TO UHT FROM TANK 02.00 MPI NET
   "S1 TOTAL STOP TANK" AT %M114.1 : Bool;   // STEP 1 TOTAL STOP TANK
   "S18 CIP TANK" AT %M120.2 : Bool;   // STEP 18 CIP
   "S24 FILLER" AT %M127.0 : Bool;   // STEP 24 FILLER
   "S35 FILLER" AT %M128.3 : Bool;   // STEP 35 FILLER
   "S47 FILLER" AT %M129.7 : Bool;   // STEP 47 FILLER
   "S9 FILLER" AT %M125.1 : Bool;   // STEP 09 FILLER
   SIP_Hamba_bit_06 AT %M151.6 : Bool;
   "ST_HEAT IP0157" AT %M138.1 : Bool;   // START HEATING FOR CIP FILLER
   StopFillers_UHT_Rec AT %M152.5 : Bool;
   "T 38 PAUSE 01.30" AT %T38 : Timer;   // PAUSE TIME AGITATOR 01.30
   "T54 LYE DOSING TOO LONG" AT %T54 : Timer;   // ACID DOSING TIME TOO LONG, SEARCH FOR FAILURE
   TIM21 AT %M61.3 : Bool;   // START TIMER 21
   TIM38 AT %M63.4 : Bool;   // START TIMER 38
   TIM55 AT %M65.5 : Bool;   // START TIMER 55
   "UPD.STEAM" AT %M86.0 : Bool;   // UPDATE STEAM TO TANK
   ViewUHT_TANK_OP25 AT %M102.7 : Bool;   // ViewUHT_TANK_OP25 ON FIXED SCREEN
   Y0108 AT %Q9.3 : Bool;   // STEAM / CIP TO VALVE 01.01
   Y0114S AT %I12.7 : Bool;   // FEEDBACK SET VALVE 01.14
   Y0143 AT %Q20.5 : Bool;   // DRAIN VALVE BOTTOM STERILE FILTER
   Y0905S AT %I44.1 : Bool;   // On off valve
   "hf ReleaseCIPfeedPump" AT %I600.5 : Bool;   // release CIP feed pump
   prF1_AhvLevel AT %QW612 : Int;   // Supplying AHV Level for IMA Hassia- Filler1
   steam_lp_request AT %I25.2 : Bool;
   "2.5Hz" AT %M10.2 : Bool;   // CYCLIC CLOCK
   "A13-DRAIN THE TANK" AT %M71.4 : Bool;   // ALARM 13
   "A30-FB FAULT VALVE 01.04" AT %M73.5 : Bool;   // ALARM 30
   "A47-FB FAULT VALVE 01.08" AT %M75.6 : Bool;   // ALARM 47
   AHV_READY AT %Q28.2 : Bool;   // AHV READY
   CIP_Hamba_bit_00 AT %M150.0 : Bool;
   "DUMMY 1 FILLING" AT %M100.0 : Bool;   // DUMMY USED IN FILLING
   "Delay De-Act V0945-SV1" AT %T76 : Timer;   // In Production relieve M0940 when stopping
   FILLER_STERILE AT %I32.3 : Bool;   // FILLER STERILE
   GS22_61 AT %I46.0 : Bool;
   "I      47.2" AT %I47.2 : Bool;
   "M19.4" AT %M19.4 : Bool;   // Filler CIP Helpbit
   MW8 AT %MW8 : Int;   // APV_Items_in_Manual_Tank
   MY0124 AT %M248.1 : Bool;   // Q 20.1; Output modul 2 Channel 1
   MY0906 AT %M252.5 : Bool;
   M_Barrier_Sterile AT %M254.3 : Bool;
   "M_Time Stop CIP" AT %M249.6 : Bool;   // Q 21.6; Output modul 2 Channel 14 was M_PACK4
   OPEN_TANK AT %I32.0 : Bool;   // OPEN BARRIER
   PROG_1_SELECTED AT %I32.6 : Bool;   // PROGRAM 1 SELECTED
   Prod_Hamba_bit_09 AT %M154.1 : Bool;
   "R.NOT USED 14" AT %M245.5 : Bool;   // RECIEVE FROM UHT MPI NET, NOT USED
   RINSE_READY AT %Q28.6 : Bool;   // RINSE READY
   "Request Drain" AT %I33.5 : Bool;   // SPARE
   "S.T.02.ALARM PULS" AT %M243.2 : Bool;   // ALARM PULS SEND TO UHT FROM TANK 02.00 MPI NET
   "S1 CHAIN WASH" AT %M137.1 : Bool;   // STEP 1 CHAIN WASH
   "S14 FILLER" AT %M125.6 : Bool;   // STEP 14 FILLER
   "S2 STOP PRODUCTION TANK" AT %M113.2 : Bool;   // STEP 2 STOP PRODUCTION TANK
   "S3 STOP CIP TANK" AT %M122.3 : Bool;   // STEP 3 STOP CIP
   "S40 FILLER" AT %M129.0 : Bool;   // STEP 40 FILLER
   "S6 PRESTERILIZING" AT %M110.6 : Bool;   // STEP 6 PRESTERILIZING TANK
   SIP_Hamba_Low_SteamPres AT %M152.1 : Bool;
   "T 31 DOSING ACID" AT %T31 : Timer;   // DOSING ACID ASEPTIC TANK
   "T 48 OPEN 01.13 CIP" AT %T48 : Timer;   // OPEN VALVE 01.13 IN CIP
   "TANK INITIALIZED" AT %M90.3 : Bool;   // TANK PLC IS INITIALIZED
   TIM14 AT %M60.4 : Bool;   // START TIMER 14
   TIM31 AT %M62.5 : Bool;   // START TIMER 31
   TIM48 AT %M64.6 : Bool;   // START TIMER 48
   TIM65 AT %M66.7 : Bool;   // START TIMER 65
   P_TT0176 AT %IW256 : Word;   // Presterilizing temperature
   "Trigger bit 3" AT %M14.2 : Bool;   // Trigger bit for calls in item control
   "UPD.TIMER 32" AT %M85.1 : Bool;   // UPDATE ACID CIRCULATION TIMER
   ValveHandling2 AT %M3.6 : Bool;   // VALVE HANDLING
   Y0101S AT %I12.0 : Bool;   // FEEDBACK SET VALVE 01.01
   Y0112R AT %I16.5 : Bool;   // FEEDBACK RESET VALVE 01.12
   Y0118 AT %Q9.5 : Bool;   // STEAM VALVE
   Y0903 AT %Q29.5 : Bool;   // High steam pressure
   Y0908 AT %Q40.4 : Bool;   // On off valve
   "hf CIPRpumpRuning" AT %I600.6 : Bool;   // CIP return pump is running
   "hf ProductRequestF1" AT %I608.0 : Bool;   // request product filler 1
   prEnableCIPValveFlipsF2 AT %Q601.3 : Bool;
   "1hz_oneshot_valve handle" AT %M4.0 : Bool;
   "A11-NOT READY FOR TOTAL" AT %M71.2 : Bool;   // ALARM 11
   "A28-FB FAULT VALVE 01.01" AT %M73.3 : Bool;   // ALARM 28
   "A45-FB FAULT VALVE 01.16" AT %M75.4 : Bool;   // ALARM 45
   AHV_HIGH_LEVEL AT %Q28.1 : Bool;   // AHV HIGH LEVEL
   CIP_FILLER_ENABLE AT %Q29.1 : Bool;   // SPARE
   CMD_AUTO AT %M3.2 : Bool;   // VALVE HANDLING
   "DUMMY2 DRAIN" AT %M99.0 : Bool;   // DUMMY DRAIN FILLING PIPE
   FILLER_ENABLE AT %I32.2 : Bool;   // FILLER CIP ENABLE
   "I      47.0" AT %I47.0 : Bool;
   "M15.0" AT %M15.0 : Bool;   // V0101 Changing
   MM0139 AT %M247.1 : Bool;   // Q 9.1; Output modul 1 Channel 9
   MY0118 AT %M247.5 : Bool;   // Q 9.5; Output modul 1 Channel 13
   MY0904 AT %M252.3 : Bool;
   M_AHV_SHUT_DOWN AT %M250.3 : Bool;   // Q 28.3; Output modul 3 Channel 3
   M_TANK_OPEN AT %M251.7 : Bool;   // Q 29.7; Output modul 3 Channel 15
   "PRODUCT_AT_TANK?" AT %I25.6 : Bool;   // PRODUCT AT TANK
   Prod_Hamba_bit_07 AT %M153.7 : Bool;
   "R.NOT USED 12" AT %M245.3 : Bool;   // RECIEVE FROM UHT MPI NET, NOT USED
   "S.T.01.TANK PRESELE." AT %M242.5 : Bool;   // TANK 1 PRESELECTED SEND TO UHT FROM TANK 01.00 MPI NET
   "S0 STOP PRODUCTION TANK" AT %M113.0 : Bool;   // MAIN FLAG STOP PRODUCTION TANK
   "S13 FILLER" AT %M125.5 : Bool;   // STEP 13 FILLER
   "S2 STOP CIP TANK" AT %M122.2 : Bool;   // STEP 2 STOP CIP
   "S3 FILLER" AT %M124.3 : Bool;   // STEP 03 FILLER
   "S4 PRESTERILIZING" AT %M110.4 : Bool;   // STEP 4 PRESTERILIZING TANK
   "S6 CIP TANK" AT %M118.6 : Bool;   // STEP 6 CIP
   "T 29 LYE CIRCULATION" AT %T29 : Timer;   // CIRCULATING LYE ASEPTIC TANK
   "T 46 PAUSE 01.13 PRES" AT %T46 : Timer;   // PAUSE TIME VALVE 01.13 IN PRESTERILIZING
   "TANK AUTO" AT %M90.0 : Bool;   // PROCESS IS RUNNING
   TIM12 AT %M60.2 : Bool;   // START TIMER 12
   TIM29 AT %M62.3 : Bool;   // START TIMER 29
   TIM46 AT %M64.4 : Bool;   // START TIMER 46
   TIM63 AT %M66.5 : Bool;   // START TIMER 63
   P_TT0160 AT %IW260 : Word;   // Steam barrier carbon filter
   "Trigger bit 1" AT %M14.0 : Bool;   // Trigger bit for calls in item control
   "UPD.TIMER 30" AT %M84.7 : Bool;   // UPDATE WATER 2 TIMER
   Y0101 AT %Q8.0 : Bool;   // PRODUCT INLET VALVE
   Y0111S AT %I12.4 : Bool;   // FEEDBACK SET VALVE 01.11
   Y0117R AT %I25.1 : Bool;   // FEEDBACK RESET VALVE 01.17
   Y0901 AT %Q29.3 : Bool;   // Low steam pressure
   Y0907R AT %I45.3 : Bool;   // On off valve
   Tag_1 AT %IW272 : Word;
   Tag_2 AT %IB274 : Byte;
   Tag_3 AT %IW275 : Word;
   Tag_4 AT %IB277 : Byte;
   Tag_5 AT %ID278 : DWord;
   Tag_6 AT %ID284 : DWord;
   Tag_7 AT %IB294 : Byte;
   Tag_8 AT %ID461 : DWord;
   Tag_9 AT %ID467 : DWord;
   Tag_10 AT %IB473 : Byte;
   Tag_11 AT %IB532 : Byte;
   Tag_12 AT %IB533 : Byte;
   Tag_13 AT %IB534 : Byte;
   Tag_14 AT %QB536 : Byte;
   Tag_15 AT %ID561 : DWord;
   Tag_16 AT %ID567 : DWord;
   Tag_17 AT %IB573 : Byte;
   Tag_18 AT %MW124 : Int;
   Tag_19 AT %MW126 : Int;
   Tag_20 AT %MW128 : Int;
   Tag_21 AT %MW110 : Int;
   Tag_22 AT %MW109 : Int;
   Tag_23 AT %MW118 : Int;
   Tag_24 AT %MW120 : Int;
   Tag_25 AT %MW122 : Int;
   Tag_26 AT %MW112 : Int;
   Tag_27 AT %MW113 : Int;
   Tag_28 AT %MW114 : Int;
   Tag_29 AT %QB535 : Byte;
   Tag_30 AT %ID600 : DWord;
   Tag_31 AT %ID604 : DWord;
   Tag_32 AT %IW608 : Word;
   Tag_33 AT %QW600 : Word;
   Tag_34 AT %QW604 : Word;
   Tag_35 AT %QW608 : Word;
   Tag_36 AT %MW140 : Int;
   Tag_37 AT %MW142 : Int;
   Tag_38 AT %MW144 : Int;
   Tag_39 AT %MW140 : Word;
END_VAR
